// TIA Portal V18 export
VAR_GLOBAL   // PLC tag table "Spare"
   Spare_DO_01 AT %Q6.6 : Bool;
   Spare_DO_02 AT %Q6.7 : Bool;
   Spare_DO_03 AT %Q7.0 : Bool;
   Not_Used_DO_01 AT %Q7.1 : Bool;
   Not_Used_DO_02 AT %Q7.2 : Bool;
   Not_Used_DO_03 AT %Q7.3 : Bool;
   Not_Used_DO_04 AT %Q7.4 : Bool;
   Not_Used_DO_05 AT %Q7.5 : Bool;
   Not_Used_DO_06 AT %Q7.6 : Bool;
   Not_Used_DO_07 AT %Q7.7 : Bool;
END_VAR
